{attribute 'qualified_only'}
{attribute 'strict'}
TYPE E_State :
(
	idle := 0,
	connect,
	sendMsg,
	receiveMsg,
	disconnect,
	error
) USINT;
END_TYPE

(* stored: Version 1.1.0.1, ProductVersion 3.1.4026.6
   DUT E_State: Id {74bbb70e-1fa3-45e2-a829-5c598ddfaccb} *)
